FUNCTION_BLOCK ABSTRACT A_Payload
VAR_INPUT
END_VAR
VAR_OUTPUT
END_VAR
VAR
END_VAR

END_FUNCTION_BLOCK

(* stored: Version 1.1.0.1, ProductVersion 3.1.4024.2
   POU A_Payload: Id {daf0f571-06aa-4ee0-992a-6cb984f34aba}, SpecialFunc None *)
